FUNCTION_BLOCK Curtain IMPLEMENTS I_Curtain
VAR
	Open_op AT%Q* : BOOL;
	Close_op AT%Q* : BOOL;

END_VAR

METHOD Close : BOOL
VAR_INPUT
	IN: BOOL;
END_VAR

IF NOT Open_op THEN
	Close_op	:=	IN;
END_IF
END_METHOD

METHOD Open : BOOL
VAR_INPUT
	IN: BOOL;
END_VAR

IF NOT Close_op THEN
	Open_op		:=	IN;
END_IF
END_METHOD

END_FUNCTION_BLOCK

(* stored: Version 1.1.0.1, ProductVersion 3.1.4024.13
   POU Curtain: Id {ca3ec28c-fda5-4d39-99fa-7f5db88fc28d}, SpecialFunc None
   Method Close: Id {37ad8b5b-8ace-4bf9-b1ba-f44bda034d06}
   Method Open: Id {ca8fbd4d-b476-43a1-a158-32c3d08cb5c1} *)
